FUNCTION_BLOCK VALVE_VIEW (* Valve Position Display *)
  (* Standard: 61499-1 *)
  (* Version 0.1, 2004-09-01, JHC, Rockwell Automation, Deleted QI,QO; initialized DIA:=0.. *)
  (* Version 0.0, 2000-05-01, JHC, Rockwell Automation *)
  (* Compiler header: package fb.rt.process; *)
  (* Compiler Java IBM VisualAge 3.0 *)
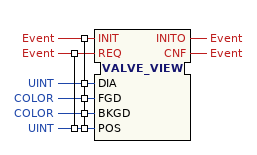
  EVENT_INPUT
    INIT WITH DIA, FGD, BKGD, POS; (* Initialization *)
    REQ WITH POS; (* Request *)
  END_EVENT
  EVENT_OUTPUT
    INITO; (* Initialization Confirm *)
    CNF; (* Service Confirmation *)
  END_EVENT
  VAR_INPUT
    DIA : UINT; (* Shaft diameter in pixels *)
    FGD : COLOR := COLOR#blue; (* Shaft body color *)
    BKGD : COLOR := COLOR#white; (* Background color *)
    POS : UINT; (* Current valve position *)
  END_VAR
END_FUNCTION_BLOCK
